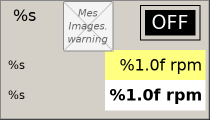
VISUALIZATION VISU_ROT  // 210x120
VAR_IN_OUT
	m_Input_ROT:		BLOCK_ROTATION_CONTINUE_ATV;
END_VAR
    RoundedRectangle (0,0 210x120)
    RoundedRectangle (145,10 50x25), "ON", invisible if: m_Input_ROT.PS.STATE_OFF
    RoundedRectangle (145,10 50x25), "OFF", invisible if: m_Input_ROT.PS.STATE_ON
    Rectangle (5,50 100x30), "%s", text list: 'TextList_Moteurs', text index: 15
    Rectangle (10,3 125x25), "%s", text variable: m_Input_ROT.PS.Mnemo, text index: 15
    RoundedRectangle (105,50 100x30), "%1.0f rpm", text variable: m_Input_ROT.PRM_Vitesse, input disabled if: NOT MACHINE.STATE_Manu
        OnMouseDown: write the text variable via InputWithLimits, min m_Input_ROT.CONF_VMIN, max m_Input_ROT.CONF_VMAX, title 'Speed'
    RoundedRectangle (105,80 100x30), "%1.0f rpm", text variable: m_Input_ROT.PS.STATE_VIT
    Image (63,1 50x50), invisible if: NOT m_Input_ROT.STATE_NOK and Not m_Input_ROT.PS.STATE_NOK, image: MesImages.warning
    RoundedRectangle (140,5 60x35), invisible if: NOT MACHINE.STATE_Manu
        tap m_Input_ROT.M_On
    Rectangle (5,80 100x30), "%s", text list: 'TextList_Moteurs', text index: 7
END_VISUALIZATION

(* stored: Version 1.1.0.1, ProductVersion 3.1.4024.6
   Visu VISU_ROT: Id {ce17fc4d-0d68-45a0-8951-58b41b1a14bc} *)
